TYPE EL3002_PDOS :
	STRUCT
		
		HwToPLC : EL3002_HWTOPLC_PDOS;
		
	END_STRUCT
END_TYPE

(* stored: Version 1.1.0.1
   DUT EL3002_PDOS: Id {76b44688-2a89-4572-b1cc-6550f5f8b520} *)
